# EPICS autosave request: andor3App/Db/andor3_settings.req
$(P)$(R)FrameRate
$(P)$(R)PreAmpGain
$(P)$(R)ReadoutRate
$(P)$(R)Overlap
$(P)$(R)NoiseFilter
$(P)$(R)PixelEncoding
$(P)$(R)A3Binning
$(P)$(R)A3ShutterMode
$(P)$(R)SensorCooling
$(P)$(R)TempControl
$(P)$(R)FanSpeed
$(P)$(R)GateMode
$(P)$(R)InsertionDelay
$(P)$(R)MCPIntelligate
$(P)$(R)MCPGain
file "ADBase_settings.req", P=$(P), R=$(R)
